{attribute 'qualified_only'}
VAR_GLOBAL
	changeAxisEnable: FB_TcMessage;
END_VAR

(* stored: Version 1.1.0.1, ProductVersion 3.1.4022.12
   GVL MSG: Id {2ed4dcf7-bf7b-405b-b02f-6fb8a15d2b9f} *)
